// TwinCAT 3 PLC project main
// ProgramVersion: 3.1.4024.0
// libraries:
//   Tc2_Standard, * (Beckhoff Automation GmbH)
//   Tc2_System, * (Beckhoff Automation GmbH)
//   Tc3_Module, * (Beckhoff Automation GmbH)
// project tree:
//   / GlobalTextList.TcGTLO, PlcTask.TcTTO, Visualization Manager.TcVMO (not stored)
//   POUs/ MAIN.TcPOU
//   VISUs/ Visu.TcVIS
// real-time tasks:
//   TASK PlcTask: cycle T#10ms, priority 20, ADS port 350

CONFIGURATION main
    RESOURCE PLC ON TwinCAT3
        TASK PlcTask(INTERVAL := T#10ms, PRIORITY := 20);
        PROGRAM MAIN WITH PlcTask : MAIN;
    END_RESOURCE
END_CONFIGURATION

// ---- POUs/MAIN.TcPOU
PROGRAM MAIN
VAR
	nGemeten AT %I* : INT;
	nGevraagd AT %I* : INT;
	bRed AT %Q* : BOOL;
	bGreen AT %Q* : BOOL;
	
	ntest : INT;
END_VAR

//Lees een fysieke potentiometer in als de variabele nGemeten en een potiometer via de visualisatie in als nGevraagd.
//Als de gemeten waarde kleiner is dan de gewenste waarde met een tolerantie van 10%, dan moet de rode lamp branden.
//Als de gemeten waarde groter is dan de gewenste waarde met een tolerantie van 10%, dan moet de groene lamp branden.

//bRed := REAL_TO_INT(nGemeten/32767.0*15.0) < nGevraagd * 0.1 OR REAL_TO_INT(nGemeten/32767.0*15.0) * 0.1 < nGevraagd;
//bGreen := REAL_TO_INT(nGemeten/32767.0*15.0) > nGevraagd * 0.1 OR REAL_TO_INT(nGemeten/32767.0*15.0) * 0.1 > nGevraagd;

bRed := REAL_TO_INT(nGemeten / 32767.0 * 15.0) < nGevraagd * 1.1 OR REAL_TO_INT(nGemeten / 32767.0 * 15.0) < nGevraagd * 0.9;
bGreen := REAL_TO_INT(nGemeten / 32767.0 * 15.0) > nGevraagd * 1.1 OR REAL_TO_INT(nGemeten / 32767.0 * 15.0) > nGevraagd * 0.9;

END_PROGRAM

// ---- GlobalTextList.TcGTLO
TEXTLIST GlobalTextList
  81 = 'Gemeten'
  734 = 'Gevraagd'
END_TEXTLIST

// ---- VISUs/Visu.TcVIS
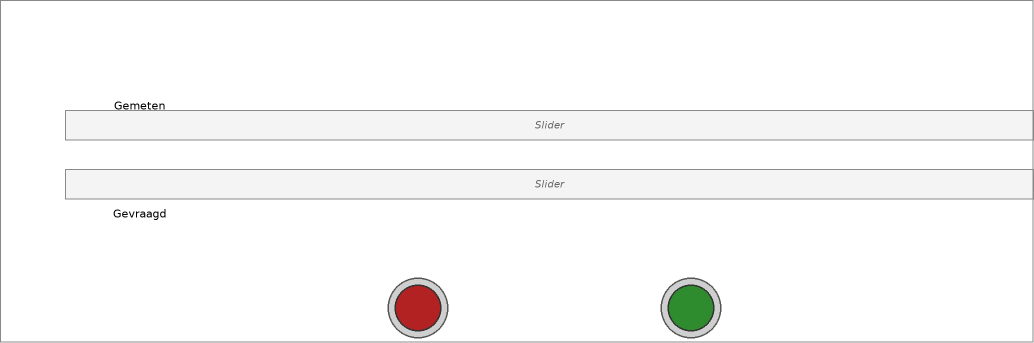
VISUALIZATION Visu  // 1034x343
    Lamp1 (656,273 70x70), variable: MAIN.bGreen, style: Lamp-Lamp1-Green
    Lamp1 (383,273 70x70), variable: MAIN.bRed, style: Lamp-Lamp1-Red
    Slider (65,110 969x30), variable: MAIN.nGemeten, scale 0..32767
    Slider (65,169 969x30), variable: MAIN.nGevraagd, scale 0..15
    Label (65,199 150x30), "Gevraagd"
    Label (65,91 150x30), "Gemeten"
END_VISUALIZATION
